FUNCTION F_GetSubsystemInterface : ST_SubsystemInterface
(**************************************************************************************
 * 	Application		:	BoxControl Framework
 *	Revision		:	$Revision: 404529 $
 *	Revision date	:	$Date: 2018-04-23 08:21:38 +0200 (Mo., 23 Apr 2018) $
 *	Last changed by	:	$Author: b7bolm $
 *	URL				:	$URL: http://almscdc.swisslog.com/repo/SWPD/Development/BoxControlFramework/20_Release/trunk/01_Software/BCF/BCF/JumpStart/20_Product/10_App/15_Subsystem/10_Lib/10_Conv/10_Functions/F_GetSubSystemInterface.TcPOU $
 *
 *	Purpose			:	Returns group interface
 *
 * ------------------------------------------------------------------------------------
 *	Copyright Swisslog [IP AG], Switzerland. All rights reserved.
 * 
 * ------------------------------------------------------------------------------------
 *	
 * 	Revision History: 
 *
 * 	VERSION			DATE			INITIALS			DESCRIPTION
 *	0.1				01.01.2001		swl					Example
 *
 **************************************************************************************)

// Get Master speed from subsystem
IF __ISVALIDREF(SubsystemRegistry.rSubsystem) THEN
	// Return Subsystem interface
	F_GetSubsystemInterface := SubsystemRegistry.rSubsystem.SubsystemInterface;
END_IF

END_FUNCTION

(* stored: Version 1.1.0.1, ProductVersion 3.1.4022.12
   POU F_GetSubSystemInterface: Id {a98fe3f0-2106-465a-a17e-3d3f83421b4e}, SpecialFunc None *)
